// TwinCAT 3 PLC project Examples
// Title: Examples
// Company: MyCompany
// ProjectVersion: 1.0.0.0
// ProgramVersion: 3.1.4023.0
// libraries:
//   Testbench, 1.0.0.0 (Zeugwerk GmbH)
// project tree:
//   Adder/ Adder.TcPOU
//   Adder/_Test/ AdderTest.TcPOU

// ---- Adder/Adder.TcPOU
FUNCTION_BLOCK Adder
VAR_INPUT
END_VAR
VAR_OUTPUT
END_VAR
VAR
END_VAR

METHOD AddInt : INT
VAR_INPUT
  value1 : INT;
  value2 : INT;
END_VAR
AddInt := value1 + value2;
END_METHOD

END_FUNCTION_BLOCK

// ---- Adder/_Test/AdderTest.TcPOU
FUNCTION_BLOCK AdderTest IMPLEMENTS Testbench.IUnitTest
VAR
  _adder : Adder;
END_VAR

METHOD Test_Add_ReturnsCorrectResult
VAR_INPUT
  assertions : Testbench.IAssertions;
END_VAR
VAR
  result : INT;
END_VAR
// arrange

// act
result := _adder.AddInt(5, 3);

// assert
assertions.EqualsInt(8, result, 'Result is correct');
END_METHOD

END_FUNCTION_BLOCK
